// TIA Portal V21 export
TYPE "Std_stTransferPackage"
   STRUCT
      iChannel { ExternalVisible := 'False'} : Int;
      iAddressedTarget { ExternalVisible := 'False'} : Int;
      iIndex { ExternalVisible := 'False'} : Int;
      iTransferValue { ExternalVisible := 'False'} : Int;
   END_STRUCT;
END_TYPE
